FUNCTION_BLOCK VacuumGripper EXTENDS BaseGripper
VAR_INPUT
END_VAR
VAR_OUTPUT
END_VAR
VAR
	//Hardware
	DI_TakenIn AT %I* : BOOL;
	DO_VacuumOn AT %Q* : BOOL;
	// Only used by PickAlpha
	VacuumHit AT %Q* : BOOL;
END_VAR

METHOD METH_Intake : BOOL
VAR_INPUT
END_VAR
DO_VacuumOn := TRUE;
END_METHOD

METHOD METH_Release : BOOL
VAR_INPUT
END_VAR
DO_VacuumOn := FALSE;
END_METHOD

METHOD METH_VacuumHitOff : BOOL
VAR_INPUT
END_VAR
VacuumHit := FALSE;
END_METHOD

METHOD METH_VacuumHitOn : BOOL
VAR_INPUT
END_VAR
VacuumHit := TRUE;
END_METHOD

PROPERTY WPTaken : BOOL
GET
// TODO - connect input correctly (probably hardware issue)
WPTaken := DI_TakenIn;
//WPTaken := DO_VacuumOn;
END_GET
END_PROPERTY

END_FUNCTION_BLOCK

(* stored: Version 1.1.0.1
   POU VacuumGripper: Id {e1824f14-fb2d-4a85-a223-2c1f3c1c8044}, SpecialFunc None
   Method METH_Intake: Id {255dd761-f5f3-40e3-8c76-b89b1d5566dc}
   Method METH_Release: Id {a48a7a99-38a4-42e2-b9f6-a996e9a43e8b}
   Method METH_VacuumHitOff: Id {665a2718-ac88-480e-8ee8-59f7fc60adf8}
   Method METH_VacuumHitOn: Id {fe78d978-41a9-4799-b6f1-096dec99e00d}
   Property WPTaken: Id {fdd6c02e-7f16-4d18-ab22-23bdb71366c2}
   Get Get: Id {4b75cd3c-7815-4c17-8aec-949da059a48d} *)
